TYPE csp_case_transport_accU_depth_enum :
(
	CSP_CASE_TRANSPORT_ACCU_DEPTH_STATUS_NOT_INITIALIZED 								:= 0,
	CSP_CASE_TRANSPORT_ACCU_DEPTH_STATUS_DISABLED 										:= 10,
	CSP_CASE_TRANSPORT_ACCU_DEPTH_STATUS_POSITION_CHECK									:= 20,
	CSP_CASE_TRANSPORT_ACCU_DEPTH_STATUS_ENABLE_REQUEST 								:= 30,
	CSP_CASE_TRANSPORT_ACCU_DEPTH_STATUS_ENABLED 										:= 40,
	CSP_CASE_TRANSPORT_ACCU_DEPTH_STATUS_PHASE_TO_MASTER								:= 45,
	CSP_CASE_TRANSPORT_ACCU_DEPTH_STATUS_GEAR_REQUEST									:= 50,
	CSP_CASE_TRANSPORT_ACCU_DEPTH_STATUS_GEARING										:= 60,
	CSP_CASE_TRANSPORT_ACCU_DEPTH_STATUS_GEARED											:= 70,
	CSP_CASE_TRANSPORT_ACCU_DEPTH_STATUS_MOVING											:= 80,
	CSP_CASE_TRANSPORT_ACCU_DEPTH_STATUS_STOP_REQUEST 									:= 110,
	CSP_CASE_TRANSPORT_ACCU_DEPTH_STATUS_DISABLE_REQUEST 								:= 120,
	CSP_CASE_TRANSPORT_ACCU_DEPTH_STATUS_DISABLING 										:= 130
) := CSP_CASE_TRANSPORT_ACCU_DEPTH_STATUS_NOT_INITIALIZED;
END_TYPE

(* stored: Version 1.1.0.1, ProductVersion 3.1.4024.3
   DUT csp_case_transport_accU_depth_enum: Id {12510b80-8268-46f7-85c9-42984d0747c6} *)
